Staubli VAL3: RobotStatus.pjx

Parameters version=s7.7.2 stackSize=5000 millimeterUnit=true
Program file=start.pgx
Program file=stop.pgx
Data file=RobotStatus.dtx
